(* IEC 61131-3 sources: horner-cscape-mcp/fixtures, 13 files *)

(* ---- valid_function.st ---- *)
FUNCTION ScaleAnalog : REAL
VAR_INPUT
    RawInput : INT;
    RawMin : INT;
    RawMax : INT;
    ScaledMin : REAL;
    ScaledMax : REAL;
END_VAR

VAR
    SpanRaw : REAL;
    SpanScaled : REAL;
    Normalized : REAL;
END_VAR

SpanRaw := INT_TO_REAL(RawMax - RawMin);
SpanScaled := ScaledMax - ScaledMin;

IF SpanRaw <> 0.0 THEN
    Normalized := INT_TO_REAL(RawInput - RawMin) / SpanRaw;
    ScaleAnalog := ScaledMin + (Normalized * SpanScaled);
ELSE
    ScaleAnalog := ScaledMin;
END_IF;

END_FUNCTION

(* ---- valid_function_block.st ---- *)
FUNCTION_BLOCK FB_Hysteresis
VAR_INPUT
    ProcessVal : REAL := 0.0;
    LowThreshold : REAL := 20.0;
    HighThreshold : REAL := 80.0;
END_VAR

VAR_OUTPUT
    OutputState : BOOL := FALSE;
END_VAR

VAR
    InternalState : BOOL := FALSE;
END_VAR

IF ProcessVal >= HighThreshold THEN
    InternalState := TRUE;
ELSIF ProcessVal <= LowThreshold THEN
    InternalState := FALSE;
END_IF;

OutputState := InternalState;

END_FUNCTION_BLOCK

(* ---- advanced_ladder_forbidden.st ---- *)
(* Attempting forbidden ladder logic construct inside project *)
PROGRAM LadderAttempt
VAR
    InputContact : BOOL := TRUE;
    CoilOutput : BOOL := FALSE;
END_VAR

RUNG 1:
---[ ]--- InputContact --- ( ) --- CoilOutput
END_RUNG

END_PROGRAM

(* ---- all_types_program.st ---- *)
(* ============================================================================
 * Program exercising all 16 specified IEC 61131-3 elementary data types:
 * BOOL, BYTE, WORD, DWORD, SINT, INT, DINT, LINT, USINT, UINT, UDINT, ULINT,
 * REAL, LREAL, TIME, STRING
 * ============================================================================ *)

PROGRAM AllTypesProgram
VAR
    (* 1. Bit strings *)
    var_bool   : BOOL := TRUE;
    var_byte   : BYTE := 16#FF;
    var_word   : WORD := 16#ABCD;
    var_dword  : DWORD := 16#12345678;

    (* 2. Signed Integers *)
    var_sint   : SINT := -128;
    var_int    : INT := -32000;
    var_dint   : DINT := -2147483648;
    var_lint   : LINT := -9223372036854775807;

    (* 3. Unsigned Integers *)
    var_usint  : USINT := 255;
    var_uint   : UINT := 65535;
    var_udint  : UDINT := 4294967295;
    var_ulint  : ULINT := 18446744073709551615;

    (* 4. Floating Point Numbers *)
    var_real   : REAL := 3.14159;
    var_lreal  : LREAL := 2.718281828459045;

    (* 5. Time and Strings *)
    var_time   : TIME := T#1h30m15s500ms;
    var_string : STRING := 'Horner Cscape IEC 61131-3 Pure Structured Text';
END_VAR

(* Logic manipulating all 16 variables *)
IF var_bool THEN
    var_byte := var_byte AND 16#0F;
    var_word := var_word OR 16#00FF;
    var_dword := var_dword XOR 16#0000FFFF;

    var_sint := var_sint + 1;
    var_int := var_int + 10;
    var_dint := var_dint + 100;
    var_lint := var_lint + 1000;

    var_usint := var_usint - 1;
    var_uint := var_uint - 10;
    var_udint := var_udint - 100;
    var_ulint := var_ulint - 1000;

    var_real := var_real * 1.5;
    var_lreal := var_lreal * 2.0;

    var_time := T#5s;
    var_string := 'Updated Status String';
END_IF;

END_PROGRAM

(* ---- complex_control_logic.st ---- *)
PROGRAM ComplexControlLogic
VAR
    StateSelector : INT := 10;
    LoopIndex : INT := 0;
    Accumulator : DINT := 0;
    ConditionMet : BOOL := FALSE;
    Buffer : ARRAY [1..10] OF INT;
    TimerDelay : TON;
    ProcessComplete : BOOL := FALSE;
END_VAR

(* 1. CASE Statement *)
CASE StateSelector OF
    0:
        Accumulator := 0;
    10:
        (* 2. FOR Loop *)
        FOR LoopIndex := 1 TO 10 DO
            Buffer[LoopIndex] := LoopIndex * 5;
            Accumulator := Accumulator + INT_TO_DINT(Buffer[LoopIndex]);
        END_FOR;
        StateSelector := 20;
    20:
        (* 3. WHILE Loop *)
        LoopIndex := 1;
        WHILE LoopIndex <= 5 DO
            Accumulator := Accumulator + INT_TO_DINT(Buffer[LoopIndex]);
            LoopIndex := LoopIndex + 1;
        END_WHILE;
        StateSelector := 30;
    30:
        (* 4. REPEAT Loop *)
        LoopIndex := 10;
        REPEAT
            Accumulator := Accumulator - 1;
            LoopIndex := LoopIndex - 1;
        UNTIL LoopIndex <= 0 END_REPEAT;
        StateSelector := 40;
    40:
        (* 5. Timer Function Block Call *)
        TimerDelay(IN := TRUE, PT := T#500ms);
        IF TimerDelay.Q THEN
            TimerDelay(IN := FALSE);
            ProcessComplete := TRUE;
            StateSelector := 0;
        END_IF;
    ELSE
        StateSelector := 0;
END_CASE;

END_PROGRAM

(* ---- mismatched_types.st ---- *)
PROGRAM MismatchedTypesProgram
VAR
    FlagBool : BOOL := FALSE;
    CounterInt : INT := 0;
    NameString : STRING := 'Test';
    TimerVal : TIME := T#1s;
END_VAR

(* Incompatible direct literal assignments *)
FlagBool := 123;
CounterInt := 'IllegalString';
CounterInt := 3.14159;
TimerVal := 500;

END_PROGRAM

(* ---- missing_semicolon.st ---- *)
PROGRAM MissingSemicolonProgram
VAR
    ValidVar : INT := 10;
    BrokenVar : BOOL := FALSE
END_VAR

ValidVar := ValidVar + 1
BrokenVar := TRUE;

END_PROGRAM

(* ---- unclosed_case.st ---- *)
PROGRAM UnclosedCaseProgram
VAR
    Selector : INT := 1;
    Result : INT := 0;
END_VAR

CASE Selector OF
    1: Result := 10;
    2: Result := 20;
(* Missing END_CASE; *)

END_PROGRAM

(* ---- unclosed_for.st ---- *)
PROGRAM UnclosedForProgram
VAR
    Index : INT := 0;
    Sum : INT := 0;
END_VAR

FOR Index := 1 TO 10 DO
    Sum := Sum + Index;
(* Missing END_FOR; *)

END_PROGRAM

(* ---- unclosed_if.st ---- *)
PROGRAM UnclosedIfProgram
VAR
    ConditionA : BOOL := TRUE;
    OutputVal : INT := 0;
END_VAR

IF ConditionA THEN
    OutputVal := 42;
(* Missing END_IF; here *)

END_PROGRAM

(* ---- unclosed_var.st ---- *)
PROGRAM UnclosedVarProgram
VAR
    A : INT := 1;
    B : INT := 2;
(* Missing END_VAR *)

A := B + 10;

END_PROGRAM

(* ---- undeclared_variable.st ---- *)
PROGRAM UndeclaredVariableProgram
VAR
    DeclaredCounter : INT := 0;
END_VAR

DeclaredCounter := DeclaredCounter + 1;
UndeclaredFlag := TRUE;
DeclaredCounter := PhantomMultiplier * 10;

END_PROGRAM

(* ---- valid_program.st ---- *)
PROGRAM SimpleProgram
VAR
    RunCommand : BOOL := FALSE;
    CycleCounter : INT := 0;
    CycleLimit : INT := 100;
    CycleComplete : BOOL := FALSE;
END_VAR

IF RunCommand THEN
    IF CycleCounter < CycleLimit THEN
        CycleCounter := CycleCounter + 1;
    ELSE
        CycleComplete := TRUE;
    END_IF;
ELSE
    CycleComplete := FALSE;
END_IF;

END_PROGRAM
